TYPE ST_AxisMap :
STRUCT
	stAxisMappingJson : ARRAY [0..67] OF  ST_AxisMapping;	
END_STRUCT
END_TYPE

(* stored: Version 1.1.0.1, ProductVersion 3.1.4024.12
   DUT ST_AxisMap: Id {790d94f2-0a53-471c-b5d6-8bb5623bdabf} *)
